FUNCTION Convert_STRING_TO_STRING : BOOL
VAR_INPUT
	in : STRING;
	out : REFERENCE TO STRING;
END_VAR

out := in;
Convert_STRING_TO_STRING := TRUE;

END_FUNCTION

(* stored: Version 1.1.0.1, ProductVersion 3.1.4024.12
   POU Convert_STRING_TO_STRING: Id {a410dc35-25c5-44f1-9fd5-46ea15a198d3}, SpecialFunc None *)
